FUNCTION f_Division : REAL
VAR_INPUT
	rDiv	:	REAL;
	rQout	:	REAL;
END_VAR
VAR
END_VAR

IF  rQout = 0 THEN
	f_Division := 0;
ELSE
	f_Division := rDiv / rQout;
END_IF

END_FUNCTION

(* stored: Version 1.1.0.1, ProductVersion 3.1.4024.12
   POU f_Division: Id {c12bb263-2327-41d7-ac4d-8f98f09d360a}, SpecialFunc None *)
